FUNCTION_BLOCK FB_ErrorHandling
VAR_INPUT
	I_bSysState		:BOOL;
	I_bReset		:BOOL;
END_VAR
VAR_OUTPUT
	O_bSysError		:BOOL;
END_VAR
VAR
	ErrorHandling	:SR;
END_VAR

ErrorHandling(SET1 := I_bSysState);

IF I_bReset THEN
	ErrorHandling.RESET := TRUE;
ELSE
	ErrorHandling.RESET := FALSE;
END_IF

O_bSysError := ErrorHandling.Q1;

END_FUNCTION_BLOCK

(* stored: Version 1.1.0.1, ProductVersion 3.1.4024.12
   POU FB_ErrorHandling: Id {b63a2be9-57a7-4fc8-bffa-deddcffa3676}, SpecialFunc None *)
